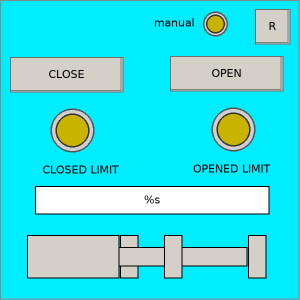
VISUALIZATION vPISTON  // 300x300
VAR_IN_OUT
	PIST1: FB_PISTON;
	MANUAL:BOOL;
	
END_VAR
    Button (170,56 113x35), "OPEN"
        OnMouseDown: execute { PIST1.bOPEN_CMD:=TRUE; }
    Rectangle (35,186 234x28), "%s", text variable: PIST1.sSTATE
    Lamp1 (47,104 51x53), variable: PIST1.bCLOSED_LIMIT, style: Lamp-Lamp1-Yellow
    Label (31,155 99x30), "CLOSED LIMIT"
    Lamp1 (208,103 51x53), variable: PIST1.bOPEN_LIMIT, style: Lamp-Lamp1-Yellow
    Label (182,154 99x30), "OPENED LIMIT"
    Button (10,57 113x35), "CLOSE"
        OnMouseDown: execute { PIST1.bOPEN_CMD:=FALSE; }
    Lamp1 (200,10 31x28), variable: PIST1.bLOCAL_MANUAL, style: Lamp-Lamp1-Yellow
    Button (255,9 35x35), "R", colour toggle: PIST1.bLOCAL_MANUAL
        tap PIST1.bLOCAL_RESET
    Rectangle (119,247 128x19), invisible if: NOT PIST1.bOPENED
    Rectangle (248,235 18x43), invisible if: NOT PIST1.bOPENED
    Rectangle (120,235 18x43), invisible if: NOT PIST1.bCLOSED
    Rectangle (78,247 92x19), invisible if: NOT PIST1.bBUSY
    Rectangle (164,235 18x43), invisible if: NOT PIST1.bBUSY
    Rectangle (27,235 92x43), colour toggle: PIST1.bERROR
    Label (125,8 99x30), "manual"
END_VISUALIZATION

(* stored: Version 1.1.0.1, ProductVersion 3.1.4024.12
   Visu vPISTON: Id {2ca2cd44-1f79-4cce-851b-f97b96892909} *)
